FUNCTION_BLOCK ABSTRACT CUBaseGround EXTENDS TcoTaskedSequencer
VAR
	_groundDone : BOOL;
END_VAR

METHOD INTERNAL CancelGround
_groundDone := FALSE;
END_METHOD

PROPERTY GroundDone : BOOL
GET
GroundDone := _groundDone;
END_GET
END_PROPERTY

END_FUNCTION_BLOCK

(* stored: Version 1.1.0.1
   POU CUBaseGround: Id {6f1d9fb3-575b-4879-af87-70bd5e814ef6}, SpecialFunc None
   Method CancelGround: Id {46466624-8a95-0eaf-1b09-e1122d31ffd8}
   Property GroundDone: Id {b43649aa-3f30-0aae-3ddc-98b2bbcd0dfa}
   Get Get: Id {09aa944f-9da0-05e5-356c-dfbcbf966722} *)
